SUBAPPLICATION Uebung_004c6 (* Toggle Flip-Flop mit IE mit BUTTON_MULTIPLE_CLICK (3-fach Klick) *)
  (* Standard: 61499-2; Description: Copyright (c) 2023 Meisterschulen am Ostbahnhof This program and the accompanying materials are made available under the terms of the Eclipse Public License 2.0 which is available at https://www.eclipse.org/legal/epl-2.0/ SPDX-License-Identifier: EPL-2.0 *)
  (* Version 1.0, 2023-10-23, Franz Höpfinger, Meisterschulen am Ostbahnhof *)
  PACKAGE Uebungen;
  IMPORT logiBUS::io::DI::logiBUS_DI::Input_I1;
  IMPORT logiBUS::io::DI::logiBUS_DI_Events::BUTTON_MULTIPLE_CLICK;
  IMPORT logiBUS::io::DQ::logiBUS_DO::Output_Q1;
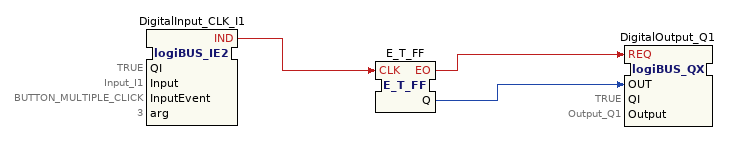
  (* Auswertung: 3-fach Klick *)
  FBS
    DigitalOutput_Q1 : logiBUS::io::DQ::logiBUS_QX(QI := TRUE, Output := Output_Q1);
    DigitalInput_CLK_I1 : logiBUS::io::DI::logiBUS_IE2(QI := TRUE, Input := Input_I1, InputEvent := BUTTON_MULTIPLE_CLICK, arg := 3);
    E_T_FF : iec61499::events::E_T_FF;
  END_FBS
  EVENT_CONNECTIONS
    DigitalInput_CLK_I1.IND TO E_T_FF.CLK;
    E_T_FF.EO TO DigitalOutput_Q1.REQ;
  END_CONNECTIONS
  DATA_CONNECTIONS
    E_T_FF.Q TO DigitalOutput_Q1.OUT;
  END_CONNECTIONS
END_SUBAPPLICATION
